{attribute 'qualified_only'}
VAR_GLOBAL
    {attribute 'pytmc' := 'pv: @(PREFIX)ARB'}
    fbArbiter: FB_Arbiter(1);
    {attribute 'pytmc' := 'pv: @(PREFIX)FFO:01'}
    fbFastFaultOutput1: FB_HardwareFFOutput := (bAutoReset := TRUE, i_sNetID := '172.21.148.161.1.1');
	{attribute 'pytmc' := 'pv: @(PREFIX)VRC:01'}
	tstVRC: FB_VRC_NO_FFO;
	
END_VAR

(* stored: Version 1.1.0.1
   GVL GVL: Id {9b9d6ea6-28e0-43fe-bc83-62be23c2a739} *)
